# EPICS substitutions: Module_11_EPICS_Device_Support/ds/dsApp/Db/user.substitutions
# Example substitutions file

file "db/dbExample1.db" {
    { user = "codac-dev" }
}

file db/dbExample2.db {
    pattern { user, no, scan }
        { "codac-dev", 1, "1 second" }
        { "codac-dev", 2, "2 second" }
        { "codac-dev", 3, "5 second" }
}
